{attribute 'GeneratedUsingTerminal: AES-D-BC-ECAT-0000'}
{attribute addProperty BoxType "AES-D-BC-ECAT-0000"}
{attribute addProperty Id "CouplerStateAT %I*UDINT4"}
{attribute addProperty CRC "3117184855"}
{attribute addProperty Size "4"}
TYPE Device_State_B9CC7757 EXTENDS TcoIo.InputBase_8311D824 :
STRUCT
	{attribute addProperty Name "CouplerState"}
	CouplerState AT %I* : UDINT;
END_STRUCT
END_TYPE

(* stored: Version 1.2.0.0, ProductVersion 3.1.4024.11
   DUT Device_State_B9CC7757: Id {66a1718b-619a-05c0-3db7-ba8d8092692f} *)
